Universal Robots PolyScope program: RC_E8_PLACE_830.urp

Program RC_E8_PLACE_830 (createdIn=3.0.0 lastSavedIn=3.0.0 directory=/programs installation=default)
Robot Program (runOnlyOnce=true motionType=MoveJ speed=1.047198 acceleration=1.396263 useActiveTCP=false)
  'Program generated by RoboDK v4.1.0 for UR3e_HORNO on 27/07/2022 12:03:21'
  'Using nominal kinematics.'
  'Using Ref. Frame Traslado C: p[0.369000, -0.220000, 0.032000, 0.000000, 0.000000, 0.000000]'
  'Using TCP 0208-0001-0001-307-000-3 Horno: p[0.000000, 0.000000, 0.038000, 0.000000, 0.000000, 0.000000]'
  Script: set_tcp(p[0.000000, 0.000000, 0.038000, 0.000000, 0.000000, 0.000000])
  Script: movej([-0.377689, -1.963670, -0.652230, -2.094395, 1.584235, 1.239184],0.60000,0.12500,0,0.0000)
  MoveL speed 100 mm/s, acceleration 120 mm/s^2 (useActiveTCP=true)
    Waypoint Waypoint_1: TCP in base x=661.848 y=-368.258 z=139.567 mm, rx=-0.0801 ry=-2.2283 rz=2.1546 rad; joints [22.21, -121.522, -108.114, -125.941, 26.026, 176.396] deg; flange x=664.331 y=-330.361 z=140.853 mm, rx=-0.0801 ry=-2.2283 rz=2.1546 rad
  'Detach from 0208-0001-0001-307-000-4 Horno'
  MoveL speed 500 mm/s, acceleration 900 mm/s^2 (useActiveTCP=true)
    Waypoint Waypoint_2: TCP in base x=658.99 y=-474.155 z=385.972 mm, rx=0.0722 ry=3.1341 rz=0.0186 rad; joints [-21.64, -112.51, -37.37, -120, 90.77, 71] deg; flange x=658.728 y=-474.601 z=423.968 mm, rx=0.0722 ry=3.1341 rz=0.0186 rad
